FUNCTION_BLOCK SOCKET
  (* Version 1.0, 2006-08-11, Goran Cengic, Chalmers *)
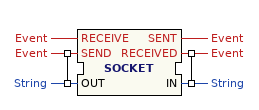
  EVENT_INPUT
    RECEIVE;
    SEND WITH OUT;
  END_EVENT
  EVENT_OUTPUT
    SENT;
    RECEIVED WITH IN;
  END_EVENT
  VAR_INPUT
    OUT : String;
  END_VAR
  VAR_OUTPUT
    IN : String;
  END_VAR
END_FUNCTION_BLOCK
